PROGRAM PRG_MainRecipe1_1
VAR
	fbrecipe		: RecipeManCommands;
	NameSave		: STRING;
	NameLoad		: STRING;
	RecipeName		: STRING;
	RecipeNameIdx	: INT;
	r1				: INT;
	dLen			: INT;
	RecipeList 		: ARRAY[0..99] OF STRING;
	tTimer			: TON;
END_VAR

PRG_RecipeList1_1();

FOR r1 := 0 TO 99 DO
	dLen 			:= LEN(PRG_RecipeList1_1.filesList[r1].sFileName) - LEN('.Recipes_2.txtrecipe'); 
	RecipeList[r1] 	:= MID(PRG_RecipeList1_1.filesList[r1].sFileName,dLen,1);
END_FOR

IF bSave2 THEN
	fbRecipe.CreateRecipe('Recipes_2',NameSave);
	PRG_RecipeList1_1.bFirst	:= TRUE;
	bSave2 					:= FALSE;
ELSIF bLoad2 THEN
	RecipeName				:= RecipeList[RecipeNameIdx];
	fbRecipe.WriteRecipe('Recipes_2', RecipeName);
	PRG_RecipeList1_1.bFirst	:= TRUE;
	bLoad2 					:= FALSE;
ELSIF bDelete2 THEN
	RecipeName				:= RecipeList[RecipeNameIdx];
	fbRecipe.DeleteRecipe('Recipes_2', RecipeName);		
	PRG_RecipeList1_1.bFirst	:= TRUE;
	bDelete2 				:= FALSE;
END_IF

END_PROGRAM

(* stored: Version 1.1.0.1, ProductVersion 3.1.4024.12
   POU PRG_MainRecipe1_1: Id {5fe8e17a-f89a-42c6-ad65-dc2b6629208d}, SpecialFunc None *)
